FUNCTION FUpdateEventTimeStampedWithSystemTimeStamepd 
VAR_INPUT
	st_event : REFERENCE TO ST_Events ;
END_VAR
VAR
	fbGetSystemTime : GETSYSTEMTIME;
	
	st_filetime : T_FILETIME;
END_VAR

fbGetSystemTime( timeLoDw => st_filetime.dwLowDateTime,
				 timeHiDW => st_filetime.dwHighDateTime);
				 
st_event.dtTimeStamped := FILETIME_TO_DT(st_filetime);

END_FUNCTION

(* stored: Version 1.1.0.1, ProductVersion 3.1.4024.12
   POU FUpdateEventTimeStampedWithSystemTimeStamepd: Id {8b4290ba-adfe-4acd-a2ff-69de9fbf2884}, SpecialFunc None *)
